// TIA Portal V17 export
// export: Created 2022-07-20T07:02:39.4346138Z, ExportSetting WithDefaults, DisplayName Totally Integrated Automation Portal, DisplayVersion V17, DisplayName TIA Portal Openness, DisplayVersion V17, DisplayName TIA Portal Version Control Interface, DisplayVersion V17, DisplayName SINAMICS Startdrive Advanced, DisplayVersion V17, DisplayName SINAMICS Startdrive G130, G150, S120, S150, SINAMICS MV, S210, DisplayVersion V17, DisplayName SINAMICS Startdrive G110M, G120, G120C, G120D, G120P, G115D, DisplayVersion V17, DisplayName STEP 7 Professional, DisplayVersion V17, DisplayName STEP 7 Safety, DisplayVersion V17, DisplayName WinCC Advanced, DisplayVersion V17
VAR_GLOBAL   // PLC tag table "LConSMC_Tags"
END_VAR
VAR_GLOBAL CONSTANT   // user constants
   LCON_ERROR_INVALID_CONFIGURATION : DWord := 16#0000_8000;
   LCON_ERROR_CYCLE_TIME_ZERO : DWord := 16#0000_8001;
   LCON_WARNING_OUTPUT_IS_LIMITED : DWord := 16#0000_4000;
   LCON_ERROR_TELEGRAM_EXTENSION : DWord := 16#0000_8002;
   LCON_ERROR_ADDITIVE_TORQUE : DWord := 16#0000_8004;
   LCON_ERROR_TORQUE_RANGE : DWord := 16#0000_8005;
   LCON_ERROR_MAX_BUFFER_SIZE_EXCEEDED : DWord := 16#0000_8006;
   LCON_WARNING_NO_VALUE_FOUND : DWord := 16#0000_4001;
   LCON_ERROR_TABLE_ENTRIES_NOT_MONOTONIC : DWord := 16#0000_8007;
   LCON_ERROR_INVALID_INPUT_PARAMETER : DWord := 16#0000_8008;
   LCON_WARNING_NO_TORQUE_PRECONTROL_ACTIVE : DWord := 16#0000_4002;
   LCON_TYPE_OF_WINDER_REWIND_FROM_ABOVE : Int := 0;   // Winder configuration parameter "TypeOfWinder"
   LCON_TYPE_OF_WINDER_REWIND_FROM_BELOW : Int := 1;   // Winder configuration parameter "TypeOfWinder"
   LCON_TYPE_OF_WINDER_UNWIND_FROM_ABOVE : Int := 2;   // Winder configuration parameter "TypeOfWinder"
   LCON_TYPE_OF_WINDER_UNWIND_FROM_BELOW : Int := 3;   // Winder configuration parameter "TypeOfWinder"
   LCON_DIAM_CALC_MODE_DIVISION : Int := 0;   // Type of diameter calculation mode
   LCON_DIAM_CALC_MODE_ADDITION : Int := 1;   // Type of diameter calculation mode
   LCON_DIAM_CALC_MODE_INTEGRAL : Int := 2;   // Type of diameter calculation mode
   LCON_DIAM_CALC_MODE_EXTERNAL : Int := 3;   // Type of diameter calculation mode
   LCON_DIAM_CALC_MODE_WEB_LENGTH : Int := 4;   // Type of diameter calculation mode
   LCON_DIAM_CALC_MODE_POSITION : Int := 5;   // Type of diameter calculation mode
   LCON_TYPE_OF_DRIVE_PULL : Int := 0;   // Section drive configuration "typeOfDrive"
   LCON_TYPE_OF_DRIVE_HELD : Int := 1;   // Section drive configuration "typeOfDrive"
   LCON_ERROR_DRIVE_DATA_ADAPTION : DWord := 16#0000_8009;
   LCON_WARNING_NO_WEB_BREAK_DETECTION_POSSIBLE : DWord := 16#0000_4003;
   LCON_ERROR_INVALID_TYPE_OF_AXIS : DWord := 16#0000_800A;
   LCON_ERROR_INVALID_DIAMETER_MODE : DWord := 16#0000_800B;
   LCON_STATEVAL_MAX_BUFFERLENGTH : UInt := 100;   // max value = 10000
   LCON_STATEVAL_MAX_BUFFERLENGTH_SUB : UInt := 10;
   LCON_STATEVAL_MAX_BUFFERLENGTH_MAIN : UInt := 100;
   LCON_TIMEPERIOD_MODE : UInt := 2;
   LCON_SAMPLEBASED_MODE : UInt := 1;
   LCON_STATEVAL_LEAST_CYCLETIME_IN_MICROSEC : UInt := 125;   // cycle time in µs
   LCON_STATEVAL_MAX_SAMPLINGRATE : UInt := 10000;   // multiple of sampling rate - do not change!
   LCON_STATEVAL_MAX_NUMBER_OF_INPUTSIGNALS : Int := 10;
   LCON_ERROR_MOVEVELOCITY : DWord := 16#0000_800C;   // Error at MC_MoveVelocity
   LCON_ERROR_INVALID_WINDERUNIT : DWord := 16#0000_800d;   // Winderunit is not rotatory
   LCON_ERROR_STOP : DWord := 16#0000_800E;   // Error at MC_Halt
   LCON_WARNING_MAXVELOCITY_EXCEEDED : DWord := 16#0000_4004;   // The configured maxVelocity has been exceeded by line- plus additionalvelocity
   LCON_MAX_VALUE_BREAK_POINT_TABLE : Int := 19;   // Maximum length of UDT LConSMC_typeBreakpointTable (0..LCON_MAX_VALUE_BREAK_POINT_TABLE)
   LCON_PI : LReal := 3.141592;
   LCON_MATERIAL_DENSITY_ACRYLONITRILE_BUTADIENE_STYRENE : LReal := 1057.2;
   LCON_MATERIAL_DENSITY_ACRYLIC : LReal := 1185.4;
   LCON_MATERIAL_DENSITY_ALUMINIUM : LReal := 2723.1;
   LCON_MATERIAL_DENSITY_CELLULOSE_ACETATE : LReal := 1297.5;
   LCON_MATERIAL_DENSITY_CELLULOSE_ACETATE_BUTYRATE : LReal := 1185.4;
   LCON_MATERIAL_DENSITY_COPPER : LReal := 8954.3;
   LCON_MATERIAL_DENSITY_CPVC : LReal := 1553.8;
   LCON_MATERIAL_DENSITY_FLUORPLASTICS : LReal := 2194.5;
   LCON_MATERIAL_DENSITY_NYLON : LReal := 1145.3;
   LCON_MATERIAL_DENSITY_PAPER : LReal := 929.1;
   LCON_MATERIAL_DENSITY_PHENOLIC : LReal := 1681.9;
   LCON_MATERIAL_DENSITY_POLYCARBONATE : LReal := 1185.4;
   LCON_MATERIAL_DENSITY_POLYESTER : LReal := 1393.6;
   LCON_MATERIAL_DENSITY_POLYETHYLENE : LReal := 961.1;
   LCON_MATERIAL_DENSITY_POLYIMIDE : LReal := 1441.7;
   LCON_MATERIAL_DENSITY_POLYPROPYLENE : LReal := 913.1;
   LCON_MATERIAL_DENSITY_POLYSTYRENE : LReal := 1057.2;
   LCON_MATERIAL_DENSITY_POLYURETHANE : LReal := 1057.2;
   LCON_MATERIAL_DENSITY_PTFE : LReal := 2194.5;
   LCON_MATERIAL_DENSITY_PVC : LReal := 1473.7;
   LCON_MATERIAL_DENSITY_STEEL : LReal := 7849.0;
   LCON_MATERIAL_DENSITY_VINYL : LReal := 1473.7;
   LCON_TAPER_NO_TAPER : Int := 0;
   LCON_TAPER_LINEAR : Int := 1;
   LCON_TAPER_HYPERBOLIC : Int := 2;
   LCON_TAPER_HYPERBOLIC_2 : Int := 3;
   LCON_TAPER_BREAKPOINT_TABLE : Int := 4;
END_VAR
